// TIA Portal V17 export
// export: Created 2024-08-09T12:52:37.2593686Z, ExportSetting WithDefaults, DisplayName Totally Integrated Automation Portal, DisplayVersion V17 Update 7, DisplayName TIA Portal Openness, DisplayVersion V17 Update 7, DisplayName TIA Portal Version Control Interface, DisplayVersion V17, DisplayName STEP 7 Professional, DisplayVersion V17 Update 7, DisplayName STEP 7 Safety, DisplayVersion V17 Update 6, DisplayName WinCC Professional, DisplayVersion V17 Update 7
DATA_BLOCK "BadgeReception3"   // DB35
{ S7_Optimized_Access := 'TRUE' }
VERSION : 0.1
// stored: AutoNumber true, DBAccessibleFromOPCUA true, DBAccessibleFromWebserver true, InstanceOfName S_Badge, InstanceOfType UDT, IsOnlyStoredInLoadMemory false, IsWriteProtectedInAS false
"S_Badge"
   // VAR RETAIN
   //    _ptmodrec : "S_REC";
   //    _PtScan : "S_Scanner";
   //    Dial_Def { S7_SetPoint := 'True'} : "S_DIALOG_DEF";
   //    _debutClignot { S7_SetPoint := 'True'} : Date_And_Time;
   //    _TpsPicke : Date_And_Time;
   //    _debutChgEtatVoyant : Date_And_Time;
   //    _TpMaintVoyant : Time;
   //    _TpClignot : Time;
   //    _DescEtp { ExternalAccessible := 'False'; ExternalVisible := 'False'; ExternalWritable := 'False'} : String[30];
   //    _CodeBadge : String[50];
   //    _NoBadgeSaisi : String;
   //    _Etp { ExternalAccessible := 'False'; ExternalVisible := 'False'; ExternalWritable := 'False'} : SInt;
   //    _Etp_Memo { ExternalAccessible := 'False'; ExternalVisible := 'False'; ExternalWritable := 'False'} : SInt;
   //    _EtpPrec { ExternalAccessible := 'False'; ExternalVisible := 'False'; ExternalWritable := 'False'} : SInt;
   //    _SvBadgeVert : Bool;
   //    _SvBadgeOrange : Bool;
   //    _SvBadgeRouge : Bool;
   //    _EtatVoyant : USInt;
   //    _FgAm : Bool;
   //    _FgBadgeSaisi : Bool;
   //    _TraitementEc : Bool;
   //    _MemoCpt { ExternalAccessible := 'False'; ExternalVisible := 'False'; ExternalWritable := 'False'} : UInt;
   //    _MemoPresence { ExternalAccessible := 'False'; ExternalVisible := 'False'; ExternalWritable := 'False'} : Bool;
   //    _FgClign : Bool;
   //    _memoEtatVoyant : USInt;
   // END_VAR
BEGIN
END_DATA_BLOCK
